FUNCTION_BLOCK setTimers (* Composite Function Block Type *)
  (* Standard: 61499-2 *)
  (* Version 0.2, 2003-12-05, JHC, Rockwell Automation, Renamed from NEWCOMPFB. *)
  (* Version 0.1, 2002-01-08, JHC, Rockwell Automation, Added DLY FB as example. *)
  (* Version 0.0, 2000-05-27, JHC, Rockwell Automation *)
  (* Compiler header: package fb.rt.template; *)
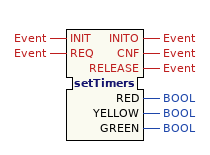
  EVENT_INPUT
    INIT; (* Initialization Request *)
    REQ; (* Normal Execution Request *)
  END_EVENT
  EVENT_OUTPUT
    INITO; (* Initialization Confirm *)
    CNF; (* Execution Confirmation *)
    RELEASE;
  END_EVENT
  VAR_OUTPUT
    RED : BOOL;
    YELLOW : BOOL;
    GREEN : BOOL;
  END_VAR
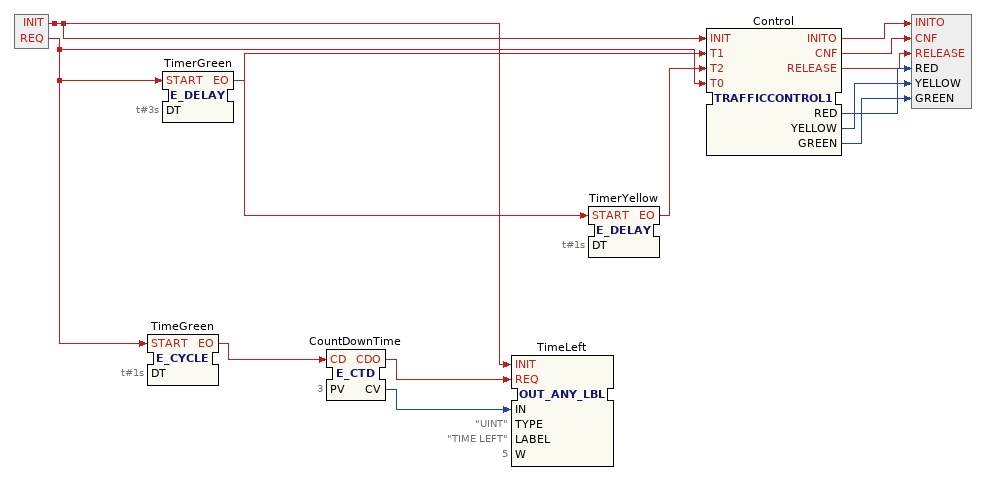
  FBS
    Control : TRAFFICCONTROL1;
    TimerGreen : E_DELAY(DT := t#3s);
    TimerYellow : E_DELAY(DT := t#1s);
    TimeGreen : E_CYCLE(DT := t#1s);
    TimeLeft : OUT_ANY_LBL(TYPE := "UINT", LABEL := "TIME LEFT", W := 5);
    CountDownTime : E_CTD(PV := 3);
  END_FBS
  EVENT_CONNECTIONS
    INIT TO Control.INIT;
    TimerGreen.EO TO Control.T1;
    TimerGreen.EO TO TimerYellow.START;
    TimerYellow.EO TO Control.T2;
    Control.INITO TO INITO;
    Control.CNF TO CNF;
    REQ TO Control.T0;
    REQ TO TimerGreen.START;
    Control.RELEASE TO RELEASE;
    REQ TO TimeGreen.START;
    INIT TO TimeLeft.INIT;
    TimeGreen.EO TO CountDownTime.CD;
    CountDownTime.CDO TO TimeLeft.REQ;
  END_CONNECTIONS
  DATA_CONNECTIONS
    Control.RED TO RED;
    Control.YELLOW TO YELLOW;
    Control.GREEN TO GREEN;
    CountDownTime.CV TO TimeLeft.IN;
  END_CONNECTIONS
END_FUNCTION_BLOCK
